(* Schneider Machine Expert - Basic project MIXER_EPP, file version 2.8.0.0 *)
(* CompanyInformations: Name=PROMASS, PhoneNumber=+39074238501, Street=Via XXV Aprile, 10/12, City=Trevi, ZipCode=06039, State=PG, Country=Italy, WebSite=www.promass.com *)
(* ProjectInformations: Name=MIXER_EPP, Description=CONTROL TO MIX-UP RECYCLED EPP (EXANDED POLYPROPILENE) WITH FRESH EPP.
AN ADDITIONAL BLOWE IS ADDED TO PERMIT THE OUTPUT FLOW *)
(* UserInformations: LastName=Torroni, FirstName=Stefano, PhoneNumber=+390742385051, Email=info@promass.com *)

HARDWARE
  Cpu 0: TM221CE16T
  EthernetConfiguration: NetworkName=M221, IpAllocationMode=FixedAddress, IpAddress=192.168.250.10, SubnetMask=255.255.255.0
  SerialLineConfiguration: Baud=Baud19200, Parity=ParityEven, DataBits=DataBits8, StopBits=StopBits1, PhysicalMedium=PhysicalMediumRs485, TransmissionMode=TransmissionModeIoScannerRtu
  MastTask: UsePeriodScanMode=false, PeriodScan=100
  FastTask: Period=255
  CpuBehavior: StartingMode=StartAutoRunForced, AutoSaveRamOnEeprom=true, WatchdogPeriod=250

SYMBOLS  (address, symbol, comment, settings)
  %M0       DRV_PWR_ON
  %M1       DRV0_JOG_INC
  %M2       DRV0_JOG_DEC
  %M3       DRV1_JOG_INC
  %M4       DRV1_JOG_DEC
  %M5       DRV0_MOVE_VEL
  %M6       DRV1_MOVE_VEL
  %M7       DRV0_ERROR
  %M8       DRV1_ERROR
  %M11      UPP_SENS_ON
  %MW0      DRV0_JOG_SPEED
  %MW1      DRV1_JOG_SPEED
  %MW2      DRV0_MOVEVEL_SPEED
  %MW3      DRV1_MOVE_VEL_SPEED
  %MW4      HMI_ALARMS
  %MW5      FSM
  %MW6      HMI_INP  "HMI>>PLC COMMANDS"
  %MW7      HMI_OUT_00  "PLC>>HMI FEEDBACK WORD 01"
  %MW8      HMI_OUT_01  "PLC>>HMI FEEDBACK WORD 02"
  %MW9      SCREW_0_RATIO
  %MW10     SCREW_1_RATIO
  %MW11     BLOWER_DELAY_OFF
  %MW12     UPP_SENS_DELAY_ON
  %TM0        [Base=OneSecond, IsDynamicPreset=true]
  %MC_JOG_ATV0   [Axis(Value(DriveAxis=DRV0)), Vel(Value(short=30))]
  %MC_JOG_ATV1   [Axis(Value(DriveAxis=DRV1)), Vel(Value(short=15))]
  %MC_MOVEVEL_ATV0   [Axis(Value(DriveAxis=DRV0)), Vel(Value(short=0))]
  %MC_MOVEVEL_ATV1   [Axis(Value(DriveAxis=DRV1)), Vel(Value(short=0))]
  %MC_POWER_ATV0   [Axis(Value(DriveAxis=DRV0))]
  %MC_POWER_ATV1   [Axis(Value(DriveAxis=DRV1))]
  %MC_READMOTIONSTATE_ATV0   [Axis(Value(DriveAxis=DRV0))]
  %MC_READMOTIONSTATE_ATV1   [Axis(Value(DriveAxis=DRV1))]
  %MC_READSTATUS_ATV0   [Axis(Value(DriveAxis=DRV0))]
  %MC_READSTATUS_ATV1   [Axis(Value(DriveAxis=DRV1))]
  %MC_RESET_ATV0   [Axis(Value(DriveAxis=DRV0))]
  %MC_RESET_ATV1   [Axis(Value(DriveAxis=DRV1))]
  %MC_STOP_ATV0   [Axis(Value(DriveAxis=DRV0))]
  %MC_STOP_ATV1   [Axis(Value(DriveAxis=DRV1))]
  %I0.0     START_BTN
  %I0.1     STOP_BTN
  %I0.2     I02
  %I0.3     QM1
  %I0.4     QM2
  %I0.5     QM3
  %I0.6     SK3
  %I0.7     MAT_LVL_UP
  %Q0.0     BLOWER

POU MAIN
  (* SectionNumber=1 *)

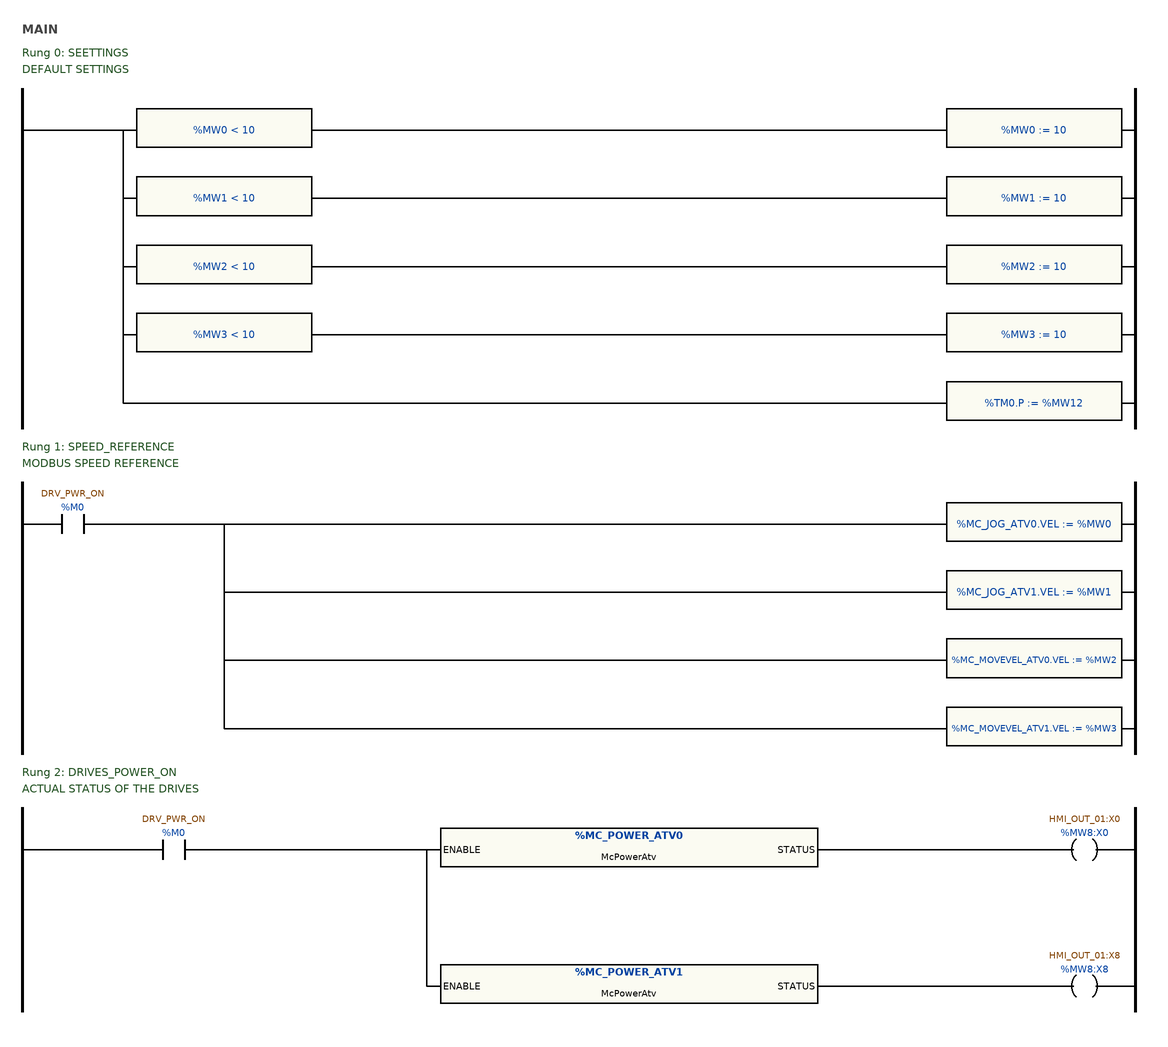

// Rung 0: SEETTINGS
// DEFAULT SETTINGS
  LD 1
  MPS
  AND [ %MW0 < 10 ]       (* DRV0_JOG_SPEED *)
  [ %MW0 := 10 ]          (* DRV0_JOG_SPEED *)
  MRD
  AND [ %MW1 < 10 ]       (* DRV1_JOG_SPEED *)
  [ %MW1 := 10 ]          (* DRV1_JOG_SPEED *)
  MRD
  AND [ %MW2 < 10 ]       (* DRV0_MOVEVEL_SPEED *)
  [ %MW2 := 10 ]          (* DRV0_MOVEVEL_SPEED *)
  MRD
  AND [ %MW3 < 10 ]       (* DRV1_MOVE_VEL_SPEED *)
  [ %MW3 := 10 ]          (* DRV1_MOVE_VEL_SPEED *)
  MPP
  [ %TM0.P := %MW12 ]     (* UPP_SENS_DELAY_ON *)
  // as ST:
  //   IF DRV0_JOG_SPEED < 10 THEN DRV0_JOG_SPEED := 10; END_IF;
  //   IF DRV1_JOG_SPEED < 10 THEN DRV1_JOG_SPEED := 10; END_IF;
  //   IF DRV0_MOVEVEL_SPEED < 10 THEN DRV0_MOVEVEL_SPEED := 10; END_IF;
  //   IF DRV1_MOVE_VEL_SPEED < 10 THEN DRV1_MOVE_VEL_SPEED := 10; END_IF;
  //   %TM0.P := UPP_SENS_DELAY_ON;

// Rung 1: SPEED_REFERENCE
// MODBUS SPEED REFERENCE
  LD %M0                  (* DRV_PWR_ON *)
  [ %MC_JOG_ATV0.VEL := %MW0 ](* DRV0_JOG_SPEED *)
  [ %MC_JOG_ATV1.VEL := %MW1 ](* DRV1_JOG_SPEED *)
  [ %MC_MOVEVEL_ATV0.VEL := %MW2 ](* DRV0_MOVEVEL_SPEED *)
  [ %MC_MOVEVEL_ATV1.VEL := %MW3 ](* DRV1_MOVE_VEL_SPEED *)
  // as ST:
  //   IF DRV_PWR_ON THEN %MC_JOG_ATV0.VEL := DRV0_JOG_SPEED; END_IF;
  //   IF DRV_PWR_ON THEN %MC_JOG_ATV1.VEL := DRV1_JOG_SPEED; END_IF;
  //   IF DRV_PWR_ON THEN %MC_MOVEVEL_ATV0.VEL := DRV0_MOVEVEL_SPEED; END_IF;
  //   IF DRV_PWR_ON THEN %MC_MOVEVEL_ATV1.VEL := DRV1_MOVE_VEL_SPEED; END_IF;

// Rung 2: DRIVES_POWER_ON
// ACTUAL STATUS OF THE DRIVES
  LD 1
  MULTIFB
  LD 1
  AND %M0                 (* DRV_PWR_ON *)
  ST %MW2009:X0
  BLK %MC_POWER_ATV0
  LD %MW2009:X0
  ENABLE
  OUT_BLK
  LD STATUS
  ST %MW8:X0              (* HMI_OUT_01 *)
  END_BLK
  BLK %MC_POWER_ATV1
  LD %MW2009:X0
  ENABLE
  OUT_BLK
  LD STATUS
  ST %MW8:X8              (* HMI_OUT_01 *)
  END_BLK
  MULTIFB
  // as ST:
  //   %MC_POWER_ATV0(ENABLE := DRV_PWR_ON);
  //   HMI_OUT_01:X0 := %MC_POWER_ATV0.STATUS;
  //   %MC_POWER_ATV1(ENABLE := DRV_PWR_ON);
  //   HMI_OUT_01:X8 := %MC_POWER_ATV1.STATUS;

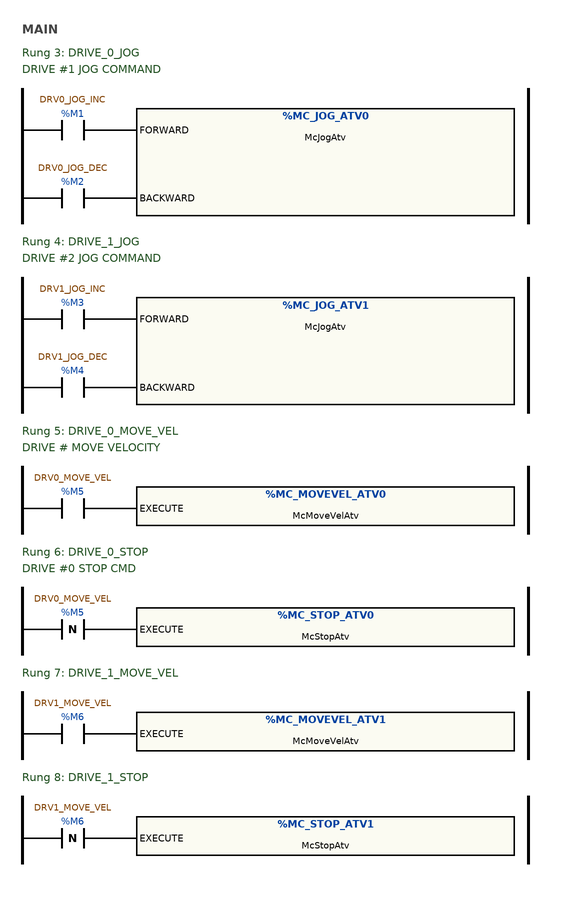

// Rung 3: DRIVE_0_JOG
// DRIVE #1 JOG COMMAND
  BLK %MC_JOG_ATV0
  LD %M1                  (* DRV0_JOG_INC *)
  FORWARD
  LD %M2                  (* DRV0_JOG_DEC *)
  BACKWARD
  END_BLK
  // as ST:
  //   %MC_JOG_ATV0(FORWARD := DRV0_JOG_INC, BACKWARD := DRV0_JOG_DEC);

// Rung 4: DRIVE_1_JOG
// DRIVE #2 JOG COMMAND
  BLK %MC_JOG_ATV1
  LD %M3                  (* DRV1_JOG_INC *)
  FORWARD
  LD %M4                  (* DRV1_JOG_DEC *)
  BACKWARD
  END_BLK
  // as ST:
  //   %MC_JOG_ATV1(FORWARD := DRV1_JOG_INC, BACKWARD := DRV1_JOG_DEC);

// Rung 5: DRIVE_0_MOVE_VEL
// DRIVE # MOVE VELOCITY
  BLK %MC_MOVEVEL_ATV0
  LD %M5                  (* DRV0_MOVE_VEL *)
  EXECUTE
  END_BLK
  // as ST:
  //   %MC_MOVEVEL_ATV0(EXECUTE := DRV0_MOVE_VEL);

// Rung 6: DRIVE_0_STOP
// DRIVE #0 STOP CMD
  BLK %MC_STOP_ATV0
  LDF %M5                 (* DRV0_MOVE_VEL *)
  EXECUTE
  END_BLK
  // as ST:
  //   %MC_STOP_ATV0(EXECUTE := FALLING(DRV0_MOVE_VEL));

// Rung 7: DRIVE_1_MOVE_VEL
  BLK %MC_MOVEVEL_ATV1
  LD %M6                  (* DRV1_MOVE_VEL *)
  EXECUTE
  END_BLK
  // as ST:
  //   %MC_MOVEVEL_ATV1(EXECUTE := DRV1_MOVE_VEL);

// Rung 8: DRIVE_1_STOP
  BLK %MC_STOP_ATV1
  LDF %M6                 (* DRV1_MOVE_VEL *)
  EXECUTE
  END_BLK
  // as ST:
  //   %MC_STOP_ATV1(EXECUTE := FALLING(DRV1_MOVE_VEL));

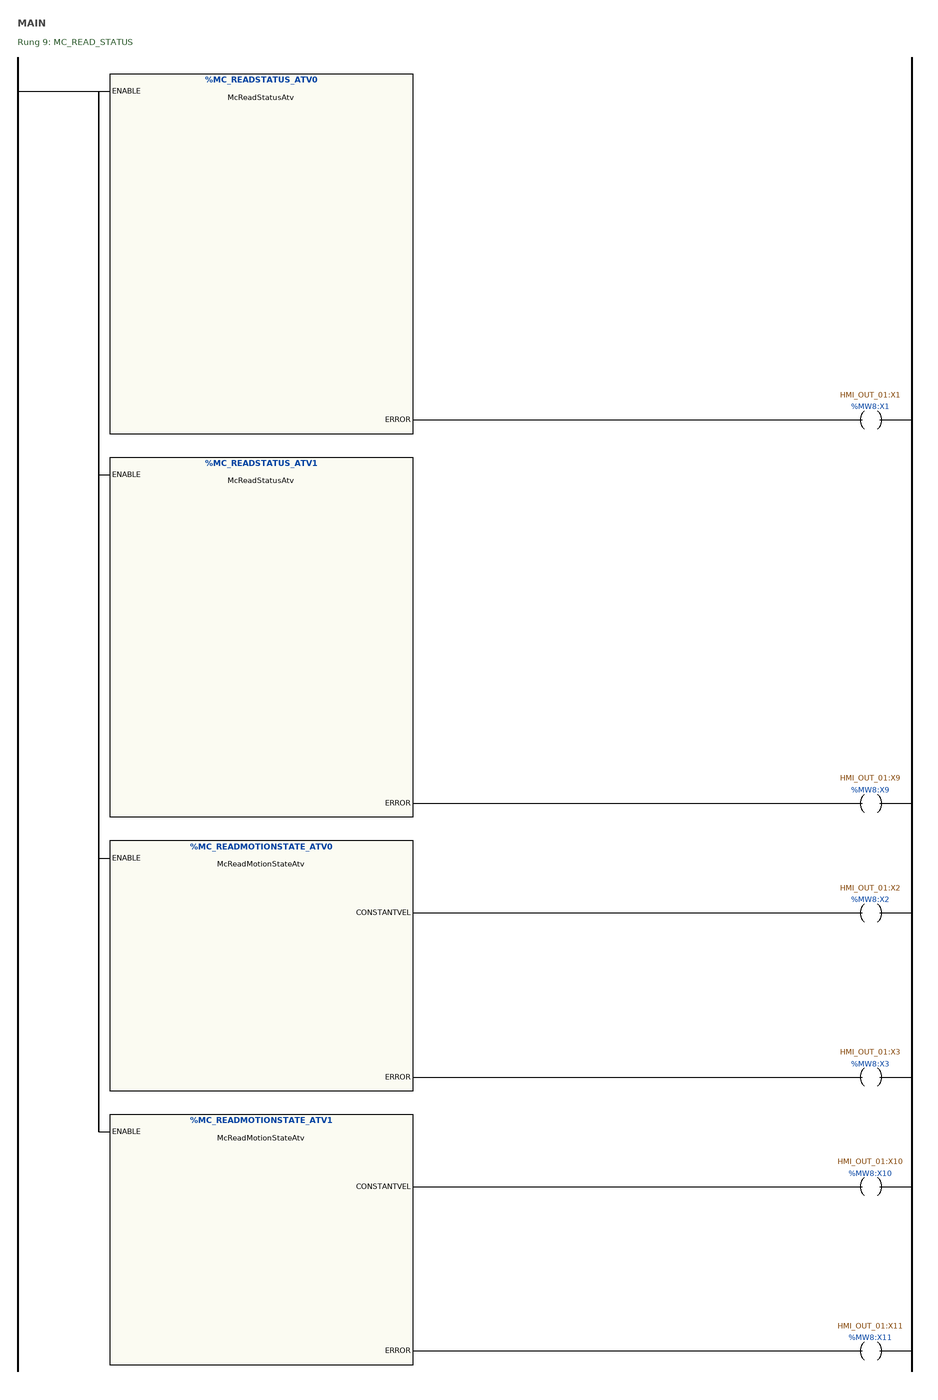

// Rung 9: MC_READ_STATUS
  LD 1
  MULTIFB
  LD 1
  ST %MW2009:X0
  BLK %MC_READSTATUS_ATV0
  LD %MW2009:X0
  ENABLE
  OUT_BLK
  LD ERROR
  ST %MW8:X1              (* HMI_OUT_01 *)
  END_BLK
  BLK %MC_READSTATUS_ATV1
  LD %MW2009:X0
  ENABLE
  OUT_BLK
  LD ERROR
  ST %MW8:X9              (* HMI_OUT_01 *)
  END_BLK
  BLK %MC_READMOTIONSTATE_ATV0
  LD %MW2009:X0
  ENABLE
  OUT_BLK
  LD CONSTANTVEL
  ST %MW8:X2              (* HMI_OUT_01 *)
  LD ERROR
  ST %MW8:X3              (* HMI_OUT_01 *)
  END_BLK
  BLK %MC_READMOTIONSTATE_ATV1
  LD %MW2009:X0
  ENABLE
  OUT_BLK
  LD CONSTANTVEL
  ST %MW8:X10             (* HMI_OUT_01 *)
  LD ERROR
  ST %MW8:X11             (* HMI_OUT_01 *)
  END_BLK
  MULTIFB
  // as ST:
  //   %MC_READSTATUS_ATV0(ENABLE := TRUE);
  //   HMI_OUT_01:X1 := %MC_READSTATUS_ATV0.ERROR;
  //   %MC_READSTATUS_ATV1(ENABLE := TRUE);
  //   HMI_OUT_01:X9 := %MC_READSTATUS_ATV1.ERROR;
  //   %MC_READMOTIONSTATE_ATV0(ENABLE := TRUE);
  //   HMI_OUT_01:X2 := %MC_READMOTIONSTATE_ATV0.CONSTANTVEL;
  //   HMI_OUT_01:X3 := %MC_READMOTIONSTATE_ATV0.ERROR;
  //   %MC_READMOTIONSTATE_ATV1(ENABLE := TRUE);
  //   HMI_OUT_01:X10 := %MC_READMOTIONSTATE_ATV1.CONSTANTVEL;
  //   HMI_OUT_01:X11 := %MC_READMOTIONSTATE_ATV1.ERROR;

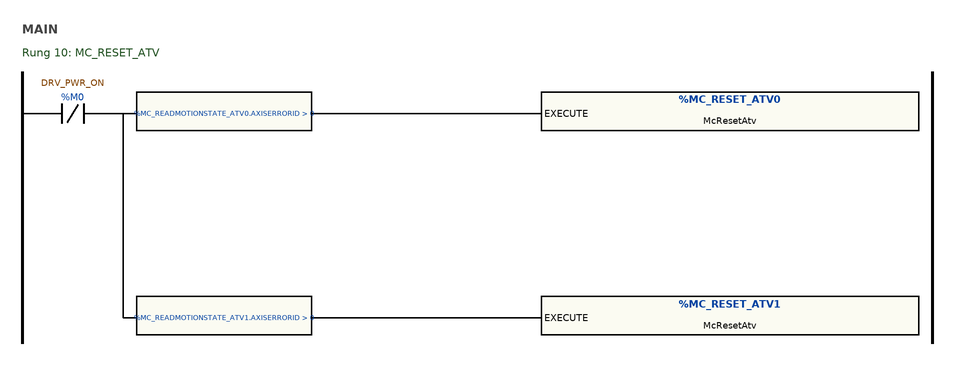

// Rung 10: MC_RESET_ATV
  LD 1
  MULTIFB
  LD 1
  ANDN %M0                (* DRV_PWR_ON *)
  ST %MW2009:X0
  BLK %MC_RESET_ATV0
  LD %MW2009:X0
  AND [ %MC_READMOTIONSTATE_ATV0.AXISERRORID > 0 ]
  EXECUTE
  END_BLK
  BLK %MC_RESET_ATV1
  LD %MW2009:X0
  AND [ %MC_READMOTIONSTATE_ATV1.AXISERRORID > 0 ]
  EXECUTE
  END_BLK
  MULTIFB
  // as ST:
  //   %MC_RESET_ATV0(EXECUTE := NOT DRV_PWR_ON AND %MC_READMOTIONSTATE_ATV0.AXISERRORID > 0);
  //   %MC_RESET_ATV1(EXECUTE := NOT DRV_PWR_ON AND %MC_READMOTIONSTATE_ATV1.AXISERRORID > 0);

POU HMI
  (* SectionNumber=2 *)

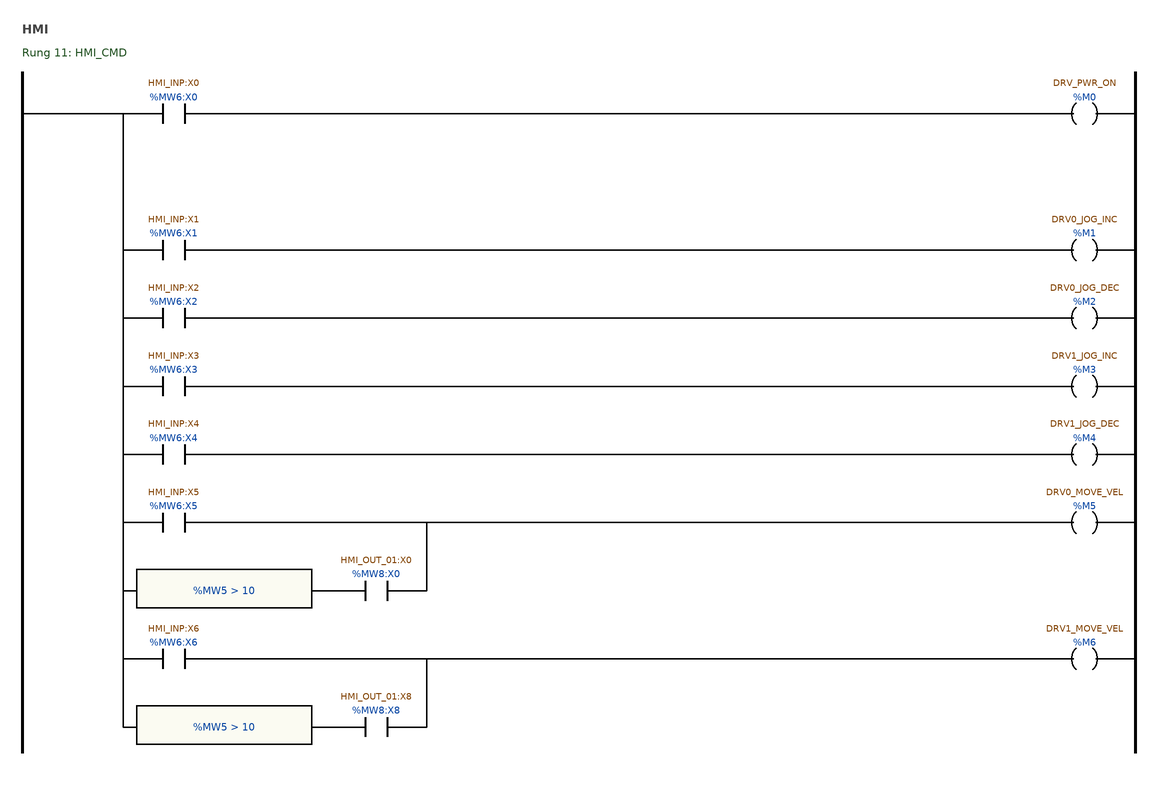

// Rung 11: HMI_CMD
  LD 1
  MPS
  AND %MW6:X0             (* HMI_INP *)
  ST %M0                  (* DRV_PWR_ON *)
  MRD
  AND %MW6:X1             (* HMI_INP *)
  ST %M1                  (* DRV0_JOG_INC *)
  MRD
  AND %MW6:X2             (* HMI_INP *)
  ST %M2                  (* DRV0_JOG_DEC *)
  MRD
  AND %MW6:X3             (* HMI_INP *)
  ST %M3                  (* DRV1_JOG_INC *)
  MRD
  AND %MW6:X4             (* HMI_INP *)
  ST %M4                  (* DRV1_JOG_DEC *)
  MRD
  AND( %MW6:X5            (* HMI_INP *)
  OR( [ %MW5 > 10 ]       (* FSM *)
  AND %MW8:X0             (* HMI_OUT_01 *)
  )
  )
  ST %M5                  (* DRV0_MOVE_VEL *)
  MPP
  AND( %MW6:X6            (* HMI_INP *)
  OR( [ %MW5 > 10 ]       (* FSM *)
  AND %MW8:X8             (* HMI_OUT_01 *)
  )
  )
  ST %M6                  (* DRV1_MOVE_VEL *)
  // as ST:
  //   DRV_PWR_ON := HMI_INP:X0;
  //   DRV0_JOG_INC := HMI_INP:X1;
  //   DRV0_JOG_DEC := HMI_INP:X2;
  //   DRV1_JOG_INC := HMI_INP:X3;
  //   DRV1_JOG_DEC := HMI_INP:X4;
  //   DRV0_MOVE_VEL := HMI_INP:X5 OR FSM > 10 AND HMI_OUT_01:X0;
  //   DRV1_MOVE_VEL := HMI_INP:X6 OR FSM > 10 AND HMI_OUT_01:X8;

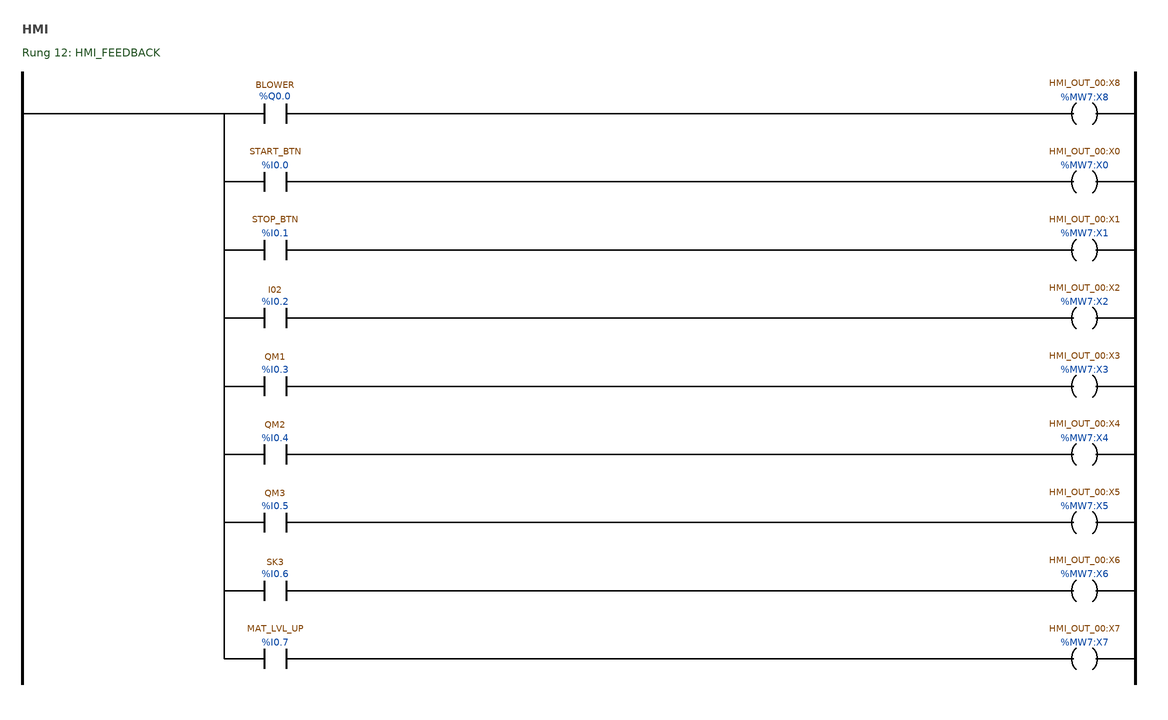

// Rung 12: HMI_FEEDBACK
  LD 1
  MPS
  AND %Q0.0               (* BLOWER *)
  ST %MW7:X8              (* HMI_OUT_00 *)
  MRD
  AND %I0.0               (* START_BTN *)
  ST %MW7:X0              (* HMI_OUT_00 *)
  MRD
  AND %I0.1               (* STOP_BTN *)
  ST %MW7:X1              (* HMI_OUT_00 *)
  MRD
  AND %I0.2               (* I02 *)
  ST %MW7:X2              (* HMI_OUT_00 *)
  MRD
  AND %I0.3               (* QM1 *)
  ST %MW7:X3              (* HMI_OUT_00 *)
  MRD
  AND %I0.4               (* QM2 *)
  ST %MW7:X4              (* HMI_OUT_00 *)
  MRD
  AND %I0.5               (* QM3 *)
  ST %MW7:X5              (* HMI_OUT_00 *)
  MRD
  AND %I0.6               (* SK3 *)
  ST %MW7:X6              (* HMI_OUT_00 *)
  MPP
  AND %I0.7               (* MAT_LVL_UP *)
  ST %MW7:X7              (* HMI_OUT_00 *)
  // as ST:
  //   HMI_OUT_00:X8 := BLOWER;
  //   HMI_OUT_00:X0 := START_BTN;
  //   HMI_OUT_00:X1 := STOP_BTN;
  //   HMI_OUT_00:X2 := I02;
  //   HMI_OUT_00:X3 := QM1;
  //   HMI_OUT_00:X4 := QM2;
  //   HMI_OUT_00:X5 := QM3;
  //   HMI_OUT_00:X6 := SK3;
  //   HMI_OUT_00:X7 := MAT_LVL_UP;

POU FSM
  (* SectionNumber=3 *)

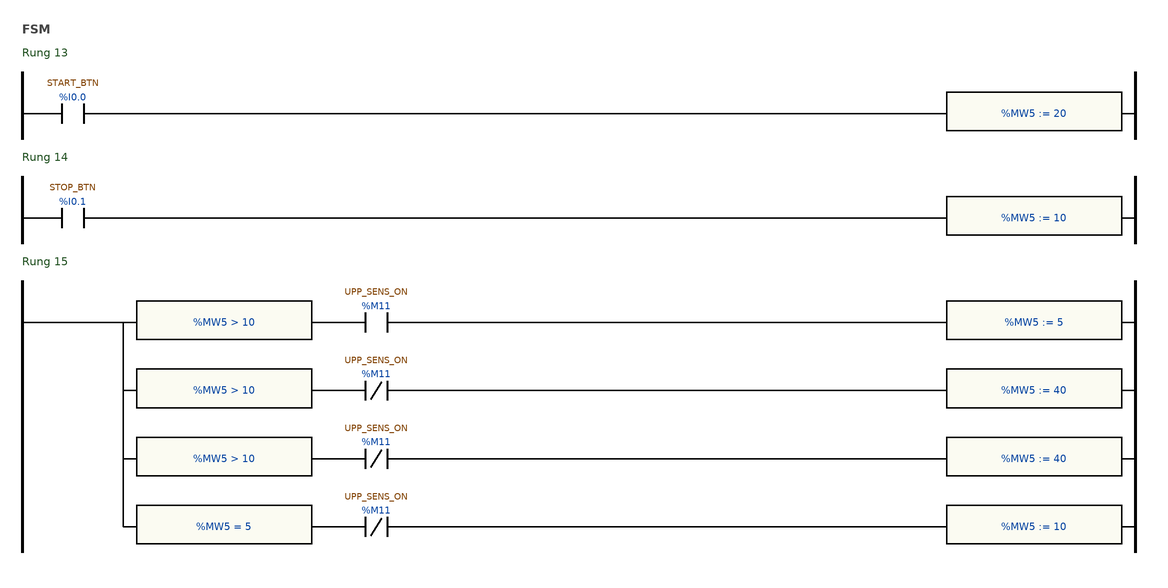

// Rung 13
  LD %I0.0                (* START_BTN *)
  [ %MW5 := 20 ]          (* FSM *)
  // as ST:
  //   IF START_BTN THEN FSM := 20; END_IF;

// Rung 14
  LD %I0.1                (* STOP_BTN *)
  [ %MW5 := 10 ]          (* FSM *)
  // as ST:
  //   IF STOP_BTN THEN FSM := 10; END_IF;

// Rung 15
  LD 1
  MPS
  AND [ %MW5 > 10 ]       (* FSM *)
  AND %M11                (* UPP_SENS_ON *)
  [ %MW5 := 5 ]           (* FSM *)
  MRD
  AND [ %MW5 > 10 ]       (* FSM *)
  ANDN %M11               (* UPP_SENS_ON *)
  [ %MW5 := 40 ]          (* FSM *)
  MRD
  AND [ %MW5 > 10 ]       (* FSM *)
  ANDN %M11               (* UPP_SENS_ON *)
  [ %MW5 := 40 ]          (* FSM *)
  MPP
  AND [ %MW5 = 5 ]        (* FSM *)
  ANDN %M11               (* UPP_SENS_ON *)
  [ %MW5 := 10 ]          (* FSM *)
  // as ST:
  //   IF FSM > 10 AND UPP_SENS_ON THEN FSM := 5; END_IF;
  //   IF FSM > 10 AND NOT UPP_SENS_ON THEN FSM := 40; END_IF;
  //   IF FSM > 10 AND NOT UPP_SENS_ON THEN FSM := 40; END_IF;
  //   IF FSM = 5 AND NOT UPP_SENS_ON THEN FSM := 10; END_IF;

POU TIMERS
  (* SectionNumber=4 *)

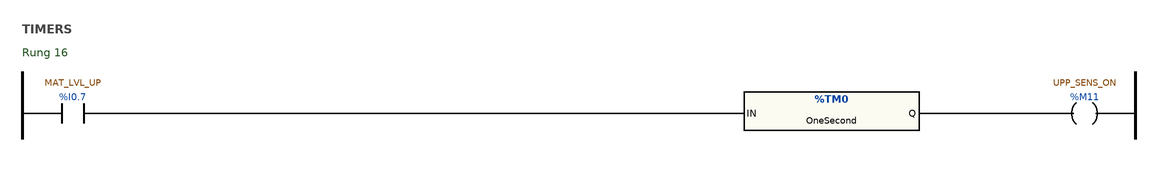

// Rung 16
  BLK %TM0
  LD %I0.7                (* MAT_LVL_UP *)
  IN
  OUT_BLK
  LD Q
  ST %M11                 (* UPP_SENS_ON *)
  END_BLK
  // as ST:
  //   %TM0(IN := MAT_LVL_UP);
  //   UPP_SENS_ON := %TM0.Q;

POU OUT
  (* SectionNumber=5 *)

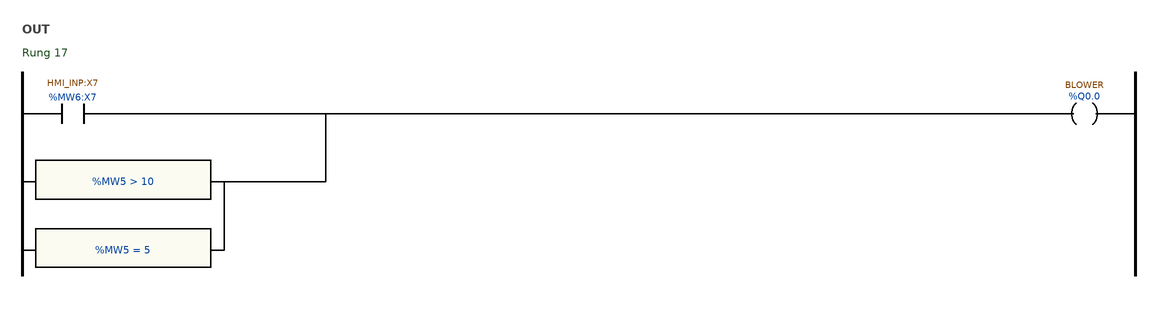

// Rung 17
  LD %MW6:X7              (* HMI_INP *)
  OR [ %MW5 > 10 ]        (* FSM *)
  OR [ %MW5 = 5 ]         (* FSM *)
  ST %Q0.0                (* BLOWER *)
  // as ST:
  //   BLOWER := HMI_INP:X7 OR FSM > 10 OR FSM = 5;
